REGION Network 132: FIXTURE IN UNIT 02 STATION 0 ANY CALIBRATION MISSING
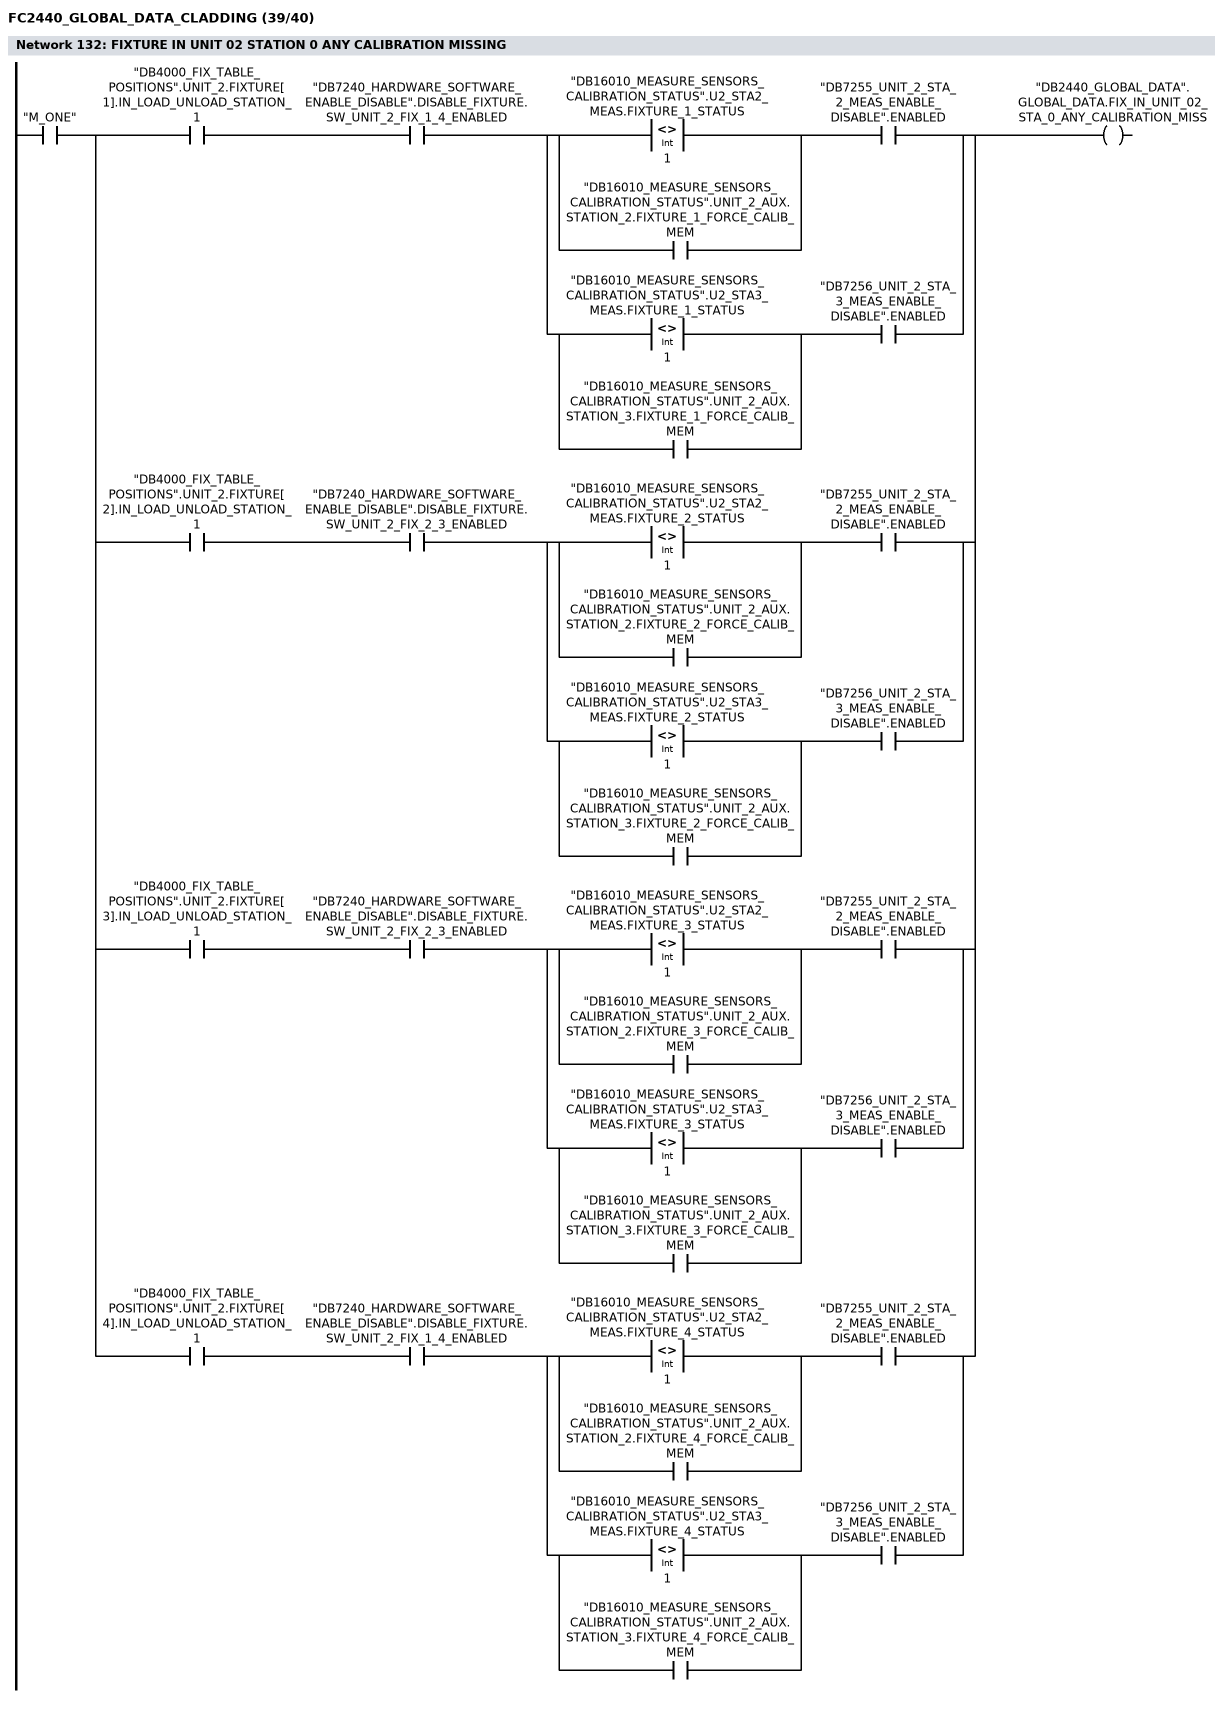
   RUNG wire#powerrail
      Contact( "M_ONE" )
      wire#w1
      Contact( "DB4000_FIX_TABLE_POSITIONS".UNIT_2.FIXTURE[1].IN_LOAD_UNLOAD_STATION_1 )
      Contact( "DB7240_HARDWARE_SOFTWARE_ENABLE_DISABLE".DISABLE_FIXTURE.SW_UNIT_2_FIX_1_4_ENABLED )
      wire#w2
      { S7_Templates := "SrcType := Int" } NE_Contact(in1 := "DB16010_MEASURE_SENSORS_CALIBRATION_STATUS".U2_STA2_MEAS.FIXTURE_1_STATUS, in2 := 1)
      wire#w3
      Contact( "DB7255_UNIT_2_STA_2_MEAS_ENABLE_DISABLE".ENABLED )
      wire#w4
      Coil( "DB2440_GLOBAL_DATA".GLOBAL_DATA.FIX_IN_UNIT_02_STA_0_ANY_CALIBRATION_MISS )
   END_RUNG
   RUNG wire#w2
      Contact( "DB16010_MEASURE_SENSORS_CALIBRATION_STATUS".UNIT_2_AUX.STATION_2.FIXTURE_1_FORCE_CALIB_MEM )
   END_RUNG wire#w3
   RUNG wire#w2
      { S7_Templates := "SrcType := Int" } NE_Contact(in1 := "DB16010_MEASURE_SENSORS_CALIBRATION_STATUS".U2_STA3_MEAS.FIXTURE_1_STATUS, in2 := 1)
      wire#w5
      Contact( "DB7256_UNIT_2_STA_3_MEAS_ENABLE_DISABLE".ENABLED )
   END_RUNG wire#w4
   RUNG wire#w2
      Contact( "DB16010_MEASURE_SENSORS_CALIBRATION_STATUS".UNIT_2_AUX.STATION_3.FIXTURE_1_FORCE_CALIB_MEM )
   END_RUNG wire#w5
   RUNG wire#w1
      Contact( "DB4000_FIX_TABLE_POSITIONS".UNIT_2.FIXTURE[2].IN_LOAD_UNLOAD_STATION_1 )
      Contact( "DB7240_HARDWARE_SOFTWARE_ENABLE_DISABLE".DISABLE_FIXTURE.SW_UNIT_2_FIX_2_3_ENABLED )
      wire#w6
      { S7_Templates := "SrcType := Int" } NE_Contact(in1 := "DB16010_MEASURE_SENSORS_CALIBRATION_STATUS".U2_STA2_MEAS.FIXTURE_2_STATUS, in2 := 1)
      wire#w7
      Contact( "DB7255_UNIT_2_STA_2_MEAS_ENABLE_DISABLE".ENABLED )
   END_RUNG wire#w4
   RUNG wire#w6
      Contact( "DB16010_MEASURE_SENSORS_CALIBRATION_STATUS".UNIT_2_AUX.STATION_2.FIXTURE_2_FORCE_CALIB_MEM )
   END_RUNG wire#w7
   RUNG wire#w6
      { S7_Templates := "SrcType := Int" } NE_Contact(in1 := "DB16010_MEASURE_SENSORS_CALIBRATION_STATUS".U2_STA3_MEAS.FIXTURE_2_STATUS, in2 := 1)
      wire#w8
      Contact( "DB7256_UNIT_2_STA_3_MEAS_ENABLE_DISABLE".ENABLED )
   END_RUNG wire#w4
   RUNG wire#w6
      Contact( "DB16010_MEASURE_SENSORS_CALIBRATION_STATUS".UNIT_2_AUX.STATION_3.FIXTURE_2_FORCE_CALIB_MEM )
   END_RUNG wire#w8
   RUNG wire#w1
      Contact( "DB4000_FIX_TABLE_POSITIONS".UNIT_2.FIXTURE[3].IN_LOAD_UNLOAD_STATION_1 )
      Contact( "DB7240_HARDWARE_SOFTWARE_ENABLE_DISABLE".DISABLE_FIXTURE.SW_UNIT_2_FIX_2_3_ENABLED )
      wire#w9
      { S7_Templates := "SrcType := Int" } NE_Contact(in1 := "DB16010_MEASURE_SENSORS_CALIBRATION_STATUS".U2_STA2_MEAS.FIXTURE_3_STATUS, in2 := 1)
      wire#w10
      Contact( "DB7255_UNIT_2_STA_2_MEAS_ENABLE_DISABLE".ENABLED )
   END_RUNG wire#w4
   RUNG wire#w9
      Contact( "DB16010_MEASURE_SENSORS_CALIBRATION_STATUS".UNIT_2_AUX.STATION_2.FIXTURE_3_FORCE_CALIB_MEM )
   END_RUNG wire#w10
   RUNG wire#w9
      { S7_Templates := "SrcType := Int" } NE_Contact(in1 := "DB16010_MEASURE_SENSORS_CALIBRATION_STATUS".U2_STA3_MEAS.FIXTURE_3_STATUS, in2 := 1)
      wire#w11
      Contact( "DB7256_UNIT_2_STA_3_MEAS_ENABLE_DISABLE".ENABLED )
   END_RUNG wire#w4
   RUNG wire#w9
      Contact( "DB16010_MEASURE_SENSORS_CALIBRATION_STATUS".UNIT_2_AUX.STATION_3.FIXTURE_3_FORCE_CALIB_MEM )
   END_RUNG wire#w11
   RUNG wire#w1
      Contact( "DB4000_FIX_TABLE_POSITIONS".UNIT_2.FIXTURE[4].IN_LOAD_UNLOAD_STATION_1 )
      Contact( "DB7240_HARDWARE_SOFTWARE_ENABLE_DISABLE".DISABLE_FIXTURE.SW_UNIT_2_FIX_1_4_ENABLED )
      wire#w12
      { S7_Templates := "SrcType := Int" } NE_Contact(in1 := "DB16010_MEASURE_SENSORS_CALIBRATION_STATUS".U2_STA2_MEAS.FIXTURE_4_STATUS, in2 := 1)
      wire#w13
      Contact( "DB7255_UNIT_2_STA_2_MEAS_ENABLE_DISABLE".ENABLED )
   END_RUNG wire#w4
   RUNG wire#w12
      Contact( "DB16010_MEASURE_SENSORS_CALIBRATION_STATUS".UNIT_2_AUX.STATION_2.FIXTURE_4_FORCE_CALIB_MEM )
   END_RUNG wire#w13
   RUNG wire#w12
      { S7_Templates := "SrcType := Int" } NE_Contact(in1 := "DB16010_MEASURE_SENSORS_CALIBRATION_STATUS".U2_STA3_MEAS.FIXTURE_4_STATUS, in2 := 1)
      wire#w14
      Contact( "DB7256_UNIT_2_STA_3_MEAS_ENABLE_DISABLE".ENABLED )
   END_RUNG wire#w4
   RUNG wire#w12
      Contact( "DB16010_MEASURE_SENSORS_CALIBRATION_STATUS".UNIT_2_AUX.STATION_3.FIXTURE_4_FORCE_CALIB_MEM )
   END_RUNG wire#w14
   // the same network as SCL:
   "DB2440_GLOBAL_DATA".GLOBAL_DATA.FIX_IN_UNIT_02_STA_0_ANY_CALIBRATION_MISS := "M_ONE" AND (("DB4000_FIX_TABLE_POSITIONS".UNIT_2.FIXTURE[1].IN_LOAD_UNLOAD_STATION_1 AND "DB7240_HARDWARE_SOFTWARE_ENABLE_DISABLE".DISABLE_FIXTURE.SW_UNIT_2_FIX_1_4_ENABLED AND (((("DB16010_MEASURE_SENSORS_CALIBRATION_STATUS".U2_STA2_MEAS.FIXTURE_1_STATUS <> 1) OR "DB16010_MEASURE_SENSORS_CALIBRATION_STATUS".UNIT_2_AUX.STATION_2.FIXTURE_1_FORCE_CALIB_MEM) AND "DB7255_UNIT_2_STA_2_MEAS_ENABLE_DISABLE".ENABLED) OR ((("DB16010_MEASURE_SENSORS_CALIBRATION_STATUS".U2_STA3_MEAS.FIXTURE_1_STATUS <> 1) OR "DB16010_MEASURE_SENSORS_CALIBRATION_STATUS".UNIT_2_AUX.STATION_3.FIXTURE_1_FORCE_CALIB_MEM) AND "DB7256_UNIT_2_STA_3_MEAS_ENABLE_DISABLE".ENABLED))) OR ("DB4000_FIX_TABLE_POSITIONS".UNIT_2.FIXTURE[2].IN_LOAD_UNLOAD_STATION_1 AND "DB7240_HARDWARE_SOFTWARE_ENABLE_DISABLE".DISABLE_FIXTURE.SW_UNIT_2_FIX_2_3_ENABLED AND (((("DB16010_MEASURE_SENSORS_CALIBRATION_STATUS".U2_STA2_MEAS.FIXTURE_2_STATUS <> 1) OR "DB16010_MEASURE_SENSORS_CALIBRATION_STATUS".UNIT_2_AUX.STATION_2.FIXTURE_2_FORCE_CALIB_MEM) AND "DB7255_UNIT_2_STA_2_MEAS_ENABLE_DISABLE".ENABLED) OR ((("DB16010_MEASURE_SENSORS_CALIBRATION_STATUS".U2_STA3_MEAS.FIXTURE_2_STATUS <> 1) OR "DB16010_MEASURE_SENSORS_CALIBRATION_STATUS".UNIT_2_AUX.STATION_3.FIXTURE_2_FORCE_CALIB_MEM) AND "DB7256_UNIT_2_STA_3_MEAS_ENABLE_DISABLE".ENABLED))) OR ("DB4000_FIX_TABLE_POSITIONS".UNIT_2.FIXTURE[3].IN_LOAD_UNLOAD_STATION_1 AND "DB7240_HARDWARE_SOFTWARE_ENABLE_DISABLE".DISABLE_FIXTURE.SW_UNIT_2_FIX_2_3_ENABLED AND (((("DB16010_MEASURE_SENSORS_CALIBRATION_STATUS".U2_STA2_MEAS.FIXTURE_3_STATUS <> 1) OR "DB16010_MEASURE_SENSORS_CALIBRATION_STATUS".UNIT_2_AUX.STATION_2.FIXTURE_3_FORCE_CALIB_MEM) AND "DB7255_UNIT_2_STA_2_MEAS_ENABLE_DISABLE".ENABLED) OR ((("DB16010_MEASURE_SENSORS_CALIBRATION_STATUS".U2_STA3_MEAS.FIXTURE_3_STATUS <> 1) OR "DB16010_MEASURE_SENSORS_CALIBRATION_STATUS".UNIT_2_AUX.STATION_3.FIXTURE_3_FORCE_CALIB_MEM) AND "DB7256_UNIT_2_STA_3_MEAS_ENABLE_DISABLE".ENABLED))) OR ("DB4000_FIX_TABLE_POSITIONS".UNIT_2.FIXTURE[4].IN_LOAD_UNLOAD_STATION_1 AND "DB7240_HARDWARE_SOFTWARE_ENABLE_DISABLE".DISABLE_FIXTURE.SW_UNIT_2_FIX_1_4_ENABLED AND (((("DB16010_MEASURE_SENSORS_CALIBRATION_STATUS".U2_STA2_MEAS.FIXTURE_4_STATUS <> 1) OR "DB16010_MEASURE_SENSORS_CALIBRATION_STATUS".UNIT_2_AUX.STATION_2.FIXTURE_4_FORCE_CALIB_MEM) AND "DB7255_UNIT_2_STA_2_MEAS_ENABLE_DISABLE".ENABLED) OR ((("DB16010_MEASURE_SENSORS_CALIBRATION_STATUS".U2_STA3_MEAS.FIXTURE_4_STATUS <> 1) OR "DB16010_MEASURE_SENSORS_CALIBRATION_STATUS".UNIT_2_AUX.STATION_3.FIXTURE_4_FORCE_CALIB_MEM) AND "DB7256_UNIT_2_STA_3_MEAS_ENABLE_DISABLE".ENABLED))));
END_REGION

REGION Network 133: UNIT 01 ANY FIXTURE CALIBRATION MISSING
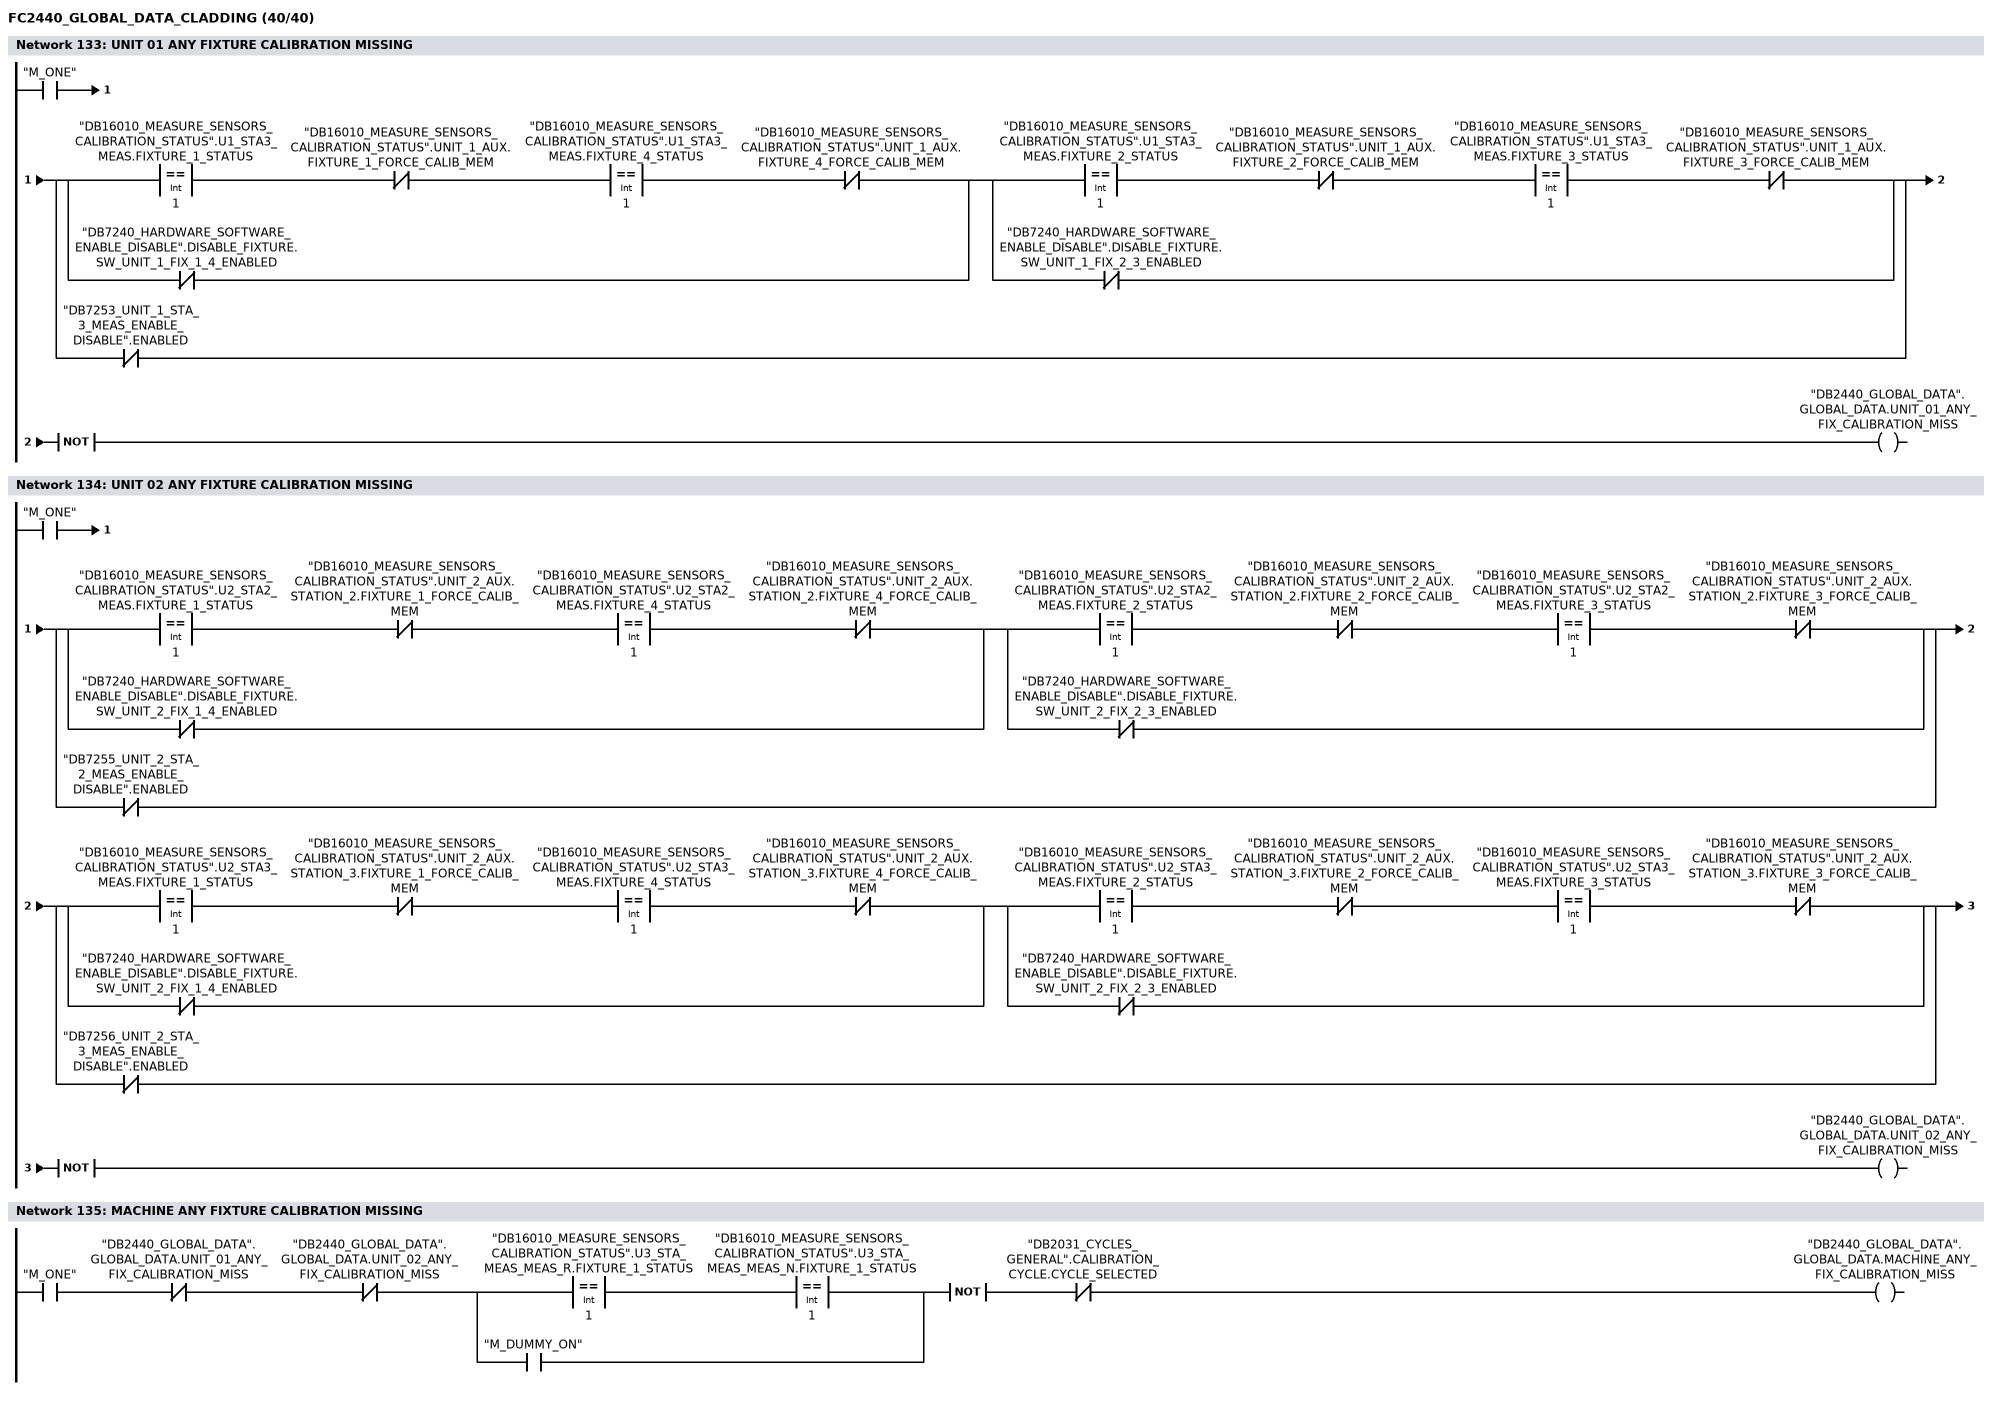
   RUNG wire#powerrail
      Contact( "M_ONE" )
      wire#w1
      { S7_Templates := "SrcType := Int" } EQ_Contact(in1 := "DB16010_MEASURE_SENSORS_CALIBRATION_STATUS".U1_STA3_MEAS.FIXTURE_1_STATUS, in2 := 1)
      I_Contact( "DB16010_MEASURE_SENSORS_CALIBRATION_STATUS".UNIT_1_AUX.FIXTURE_1_FORCE_CALIB_MEM )
      { S7_Templates := "SrcType := Int" } EQ_Contact(in1 := "DB16010_MEASURE_SENSORS_CALIBRATION_STATUS".U1_STA3_MEAS.FIXTURE_4_STATUS, in2 := 1)
      I_Contact( "DB16010_MEASURE_SENSORS_CALIBRATION_STATUS".UNIT_1_AUX.FIXTURE_4_FORCE_CALIB_MEM )
      wire#w2
      { S7_Templates := "SrcType := Int" } EQ_Contact(in1 := "DB16010_MEASURE_SENSORS_CALIBRATION_STATUS".U1_STA3_MEAS.FIXTURE_2_STATUS, in2 := 1)
      I_Contact( "DB16010_MEASURE_SENSORS_CALIBRATION_STATUS".UNIT_1_AUX.FIXTURE_2_FORCE_CALIB_MEM )
      { S7_Templates := "SrcType := Int" } EQ_Contact(in1 := "DB16010_MEASURE_SENSORS_CALIBRATION_STATUS".U1_STA3_MEAS.FIXTURE_3_STATUS, in2 := 1)
      I_Contact( "DB16010_MEASURE_SENSORS_CALIBRATION_STATUS".UNIT_1_AUX.FIXTURE_3_FORCE_CALIB_MEM )
      wire#w3
      Not()
      Coil( "DB2440_GLOBAL_DATA".GLOBAL_DATA.UNIT_01_ANY_FIX_CALIBRATION_MISS )
   END_RUNG
   RUNG wire#w1
      I_Contact( "DB7240_HARDWARE_SOFTWARE_ENABLE_DISABLE".DISABLE_FIXTURE.SW_UNIT_1_FIX_1_4_ENABLED )
   END_RUNG wire#w2
   RUNG wire#w2
      I_Contact( "DB7240_HARDWARE_SOFTWARE_ENABLE_DISABLE".DISABLE_FIXTURE.SW_UNIT_1_FIX_2_3_ENABLED )
   END_RUNG wire#w3
   RUNG wire#w1
      I_Contact( "DB7253_UNIT_1_STA_3_MEAS_ENABLE_DISABLE".ENABLED )
   END_RUNG wire#w3
   // the same network as SCL:
   "DB2440_GLOBAL_DATA".GLOBAL_DATA.UNIT_01_ANY_FIX_CALIBRATION_MISS := NOT ("M_ONE" AND ((((("DB16010_MEASURE_SENSORS_CALIBRATION_STATUS".U1_STA3_MEAS.FIXTURE_1_STATUS = 1) AND NOT "DB16010_MEASURE_SENSORS_CALIBRATION_STATUS".UNIT_1_AUX.FIXTURE_1_FORCE_CALIB_MEM AND ("DB16010_MEASURE_SENSORS_CALIBRATION_STATUS".U1_STA3_MEAS.FIXTURE_4_STATUS = 1) AND NOT "DB16010_MEASURE_SENSORS_CALIBRATION_STATUS".UNIT_1_AUX.FIXTURE_4_FORCE_CALIB_MEM) OR NOT "DB7240_HARDWARE_SOFTWARE_ENABLE_DISABLE".DISABLE_FIXTURE.SW_UNIT_1_FIX_1_4_ENABLED) AND ((("DB16010_MEASURE_SENSORS_CALIBRATION_STATUS".U1_STA3_MEAS.FIXTURE_2_STATUS = 1) AND NOT "DB16010_MEASURE_SENSORS_CALIBRATION_STATUS".UNIT_1_AUX.FIXTURE_2_FORCE_CALIB_MEM AND ("DB16010_MEASURE_SENSORS_CALIBRATION_STATUS".U1_STA3_MEAS.FIXTURE_3_STATUS = 1) AND NOT "DB16010_MEASURE_SENSORS_CALIBRATION_STATUS".UNIT_1_AUX.FIXTURE_3_FORCE_CALIB_MEM) OR NOT "DB7240_HARDWARE_SOFTWARE_ENABLE_DISABLE".DISABLE_FIXTURE.SW_UNIT_1_FIX_2_3_ENABLED)) OR NOT "DB7253_UNIT_1_STA_3_MEAS_ENABLE_DISABLE".ENABLED));
END_REGION

REGION Network 134: UNIT 02 ANY FIXTURE CALIBRATION MISSING
   RUNG wire#powerrail
      Contact( "M_ONE" )
      wire#w1
      { S7_Templates := "SrcType := Int" } EQ_Contact(in1 := "DB16010_MEASURE_SENSORS_CALIBRATION_STATUS".U2_STA2_MEAS.FIXTURE_1_STATUS, in2 := 1)
      I_Contact( "DB16010_MEASURE_SENSORS_CALIBRATION_STATUS".UNIT_2_AUX.STATION_2.FIXTURE_1_FORCE_CALIB_MEM )
      { S7_Templates := "SrcType := Int" } EQ_Contact(in1 := "DB16010_MEASURE_SENSORS_CALIBRATION_STATUS".U2_STA2_MEAS.FIXTURE_4_STATUS, in2 := 1)
      I_Contact( "DB16010_MEASURE_SENSORS_CALIBRATION_STATUS".UNIT_2_AUX.STATION_2.FIXTURE_4_FORCE_CALIB_MEM )
      wire#w2
      { S7_Templates := "SrcType := Int" } EQ_Contact(in1 := "DB16010_MEASURE_SENSORS_CALIBRATION_STATUS".U2_STA2_MEAS.FIXTURE_2_STATUS, in2 := 1)
      I_Contact( "DB16010_MEASURE_SENSORS_CALIBRATION_STATUS".UNIT_2_AUX.STATION_2.FIXTURE_2_FORCE_CALIB_MEM )
      { S7_Templates := "SrcType := Int" } EQ_Contact(in1 := "DB16010_MEASURE_SENSORS_CALIBRATION_STATUS".U2_STA2_MEAS.FIXTURE_3_STATUS, in2 := 1)
      I_Contact( "DB16010_MEASURE_SENSORS_CALIBRATION_STATUS".UNIT_2_AUX.STATION_2.FIXTURE_3_FORCE_CALIB_MEM )
      wire#w3
      { S7_Templates := "SrcType := Int" } EQ_Contact(in1 := "DB16010_MEASURE_SENSORS_CALIBRATION_STATUS".U2_STA3_MEAS.FIXTURE_1_STATUS, in2 := 1)
      I_Contact( "DB16010_MEASURE_SENSORS_CALIBRATION_STATUS".UNIT_2_AUX.STATION_3.FIXTURE_1_FORCE_CALIB_MEM )
      { S7_Templates := "SrcType := Int" } EQ_Contact(in1 := "DB16010_MEASURE_SENSORS_CALIBRATION_STATUS".U2_STA3_MEAS.FIXTURE_4_STATUS, in2 := 1)
      I_Contact( "DB16010_MEASURE_SENSORS_CALIBRATION_STATUS".UNIT_2_AUX.STATION_3.FIXTURE_4_FORCE_CALIB_MEM )
      wire#w4
      { S7_Templates := "SrcType := Int" } EQ_Contact(in1 := "DB16010_MEASURE_SENSORS_CALIBRATION_STATUS".U2_STA3_MEAS.FIXTURE_2_STATUS, in2 := 1)
      I_Contact( "DB16010_MEASURE_SENSORS_CALIBRATION_STATUS".UNIT_2_AUX.STATION_3.FIXTURE_2_FORCE_CALIB_MEM )
      { S7_Templates := "SrcType := Int" } EQ_Contact(in1 := "DB16010_MEASURE_SENSORS_CALIBRATION_STATUS".U2_STA3_MEAS.FIXTURE_3_STATUS, in2 := 1)
      I_Contact( "DB16010_MEASURE_SENSORS_CALIBRATION_STATUS".UNIT_2_AUX.STATION_3.FIXTURE_3_FORCE_CALIB_MEM )
      wire#w5
      Not()
      Coil( "DB2440_GLOBAL_DATA".GLOBAL_DATA.UNIT_02_ANY_FIX_CALIBRATION_MISS )
   END_RUNG
   RUNG wire#w1
      I_Contact( "DB7240_HARDWARE_SOFTWARE_ENABLE_DISABLE".DISABLE_FIXTURE.SW_UNIT_2_FIX_1_4_ENABLED )
   END_RUNG wire#w2
   RUNG wire#w2
      I_Contact( "DB7240_HARDWARE_SOFTWARE_ENABLE_DISABLE".DISABLE_FIXTURE.SW_UNIT_2_FIX_2_3_ENABLED )
   END_RUNG wire#w3
   RUNG wire#w1
      I_Contact( "DB7255_UNIT_2_STA_2_MEAS_ENABLE_DISABLE".ENABLED )
   END_RUNG wire#w3
   RUNG wire#w3
      I_Contact( "DB7240_HARDWARE_SOFTWARE_ENABLE_DISABLE".DISABLE_FIXTURE.SW_UNIT_2_FIX_1_4_ENABLED )
   END_RUNG wire#w4
   RUNG wire#w4
      I_Contact( "DB7240_HARDWARE_SOFTWARE_ENABLE_DISABLE".DISABLE_FIXTURE.SW_UNIT_2_FIX_2_3_ENABLED )
   END_RUNG wire#w5
   RUNG wire#w3
      I_Contact( "DB7256_UNIT_2_STA_3_MEAS_ENABLE_DISABLE".ENABLED )
   END_RUNG wire#w5
   // the same network as SCL:
   "DB2440_GLOBAL_DATA".GLOBAL_DATA.UNIT_02_ANY_FIX_CALIBRATION_MISS := NOT ("M_ONE" AND ((((("DB16010_MEASURE_SENSORS_CALIBRATION_STATUS".U2_STA2_MEAS.FIXTURE_1_STATUS = 1) AND NOT "DB16010_MEASURE_SENSORS_CALIBRATION_STATUS".UNIT_2_AUX.STATION_2.FIXTURE_1_FORCE_CALIB_MEM AND ("DB16010_MEASURE_SENSORS_CALIBRATION_STATUS".U2_STA2_MEAS.FIXTURE_4_STATUS = 1) AND NOT "DB16010_MEASURE_SENSORS_CALIBRATION_STATUS".UNIT_2_AUX.STATION_2.FIXTURE_4_FORCE_CALIB_MEM) OR NOT "DB7240_HARDWARE_SOFTWARE_ENABLE_DISABLE".DISABLE_FIXTURE.SW_UNIT_2_FIX_1_4_ENABLED) AND ((("DB16010_MEASURE_SENSORS_CALIBRATION_STATUS".U2_STA2_MEAS.FIXTURE_2_STATUS = 1) AND NOT "DB16010_MEASURE_SENSORS_CALIBRATION_STATUS".UNIT_2_AUX.STATION_2.FIXTURE_2_FORCE_CALIB_MEM AND ("DB16010_MEASURE_SENSORS_CALIBRATION_STATUS".U2_STA2_MEAS.FIXTURE_3_STATUS = 1) AND NOT "DB16010_MEASURE_SENSORS_CALIBRATION_STATUS".UNIT_2_AUX.STATION_2.FIXTURE_3_FORCE_CALIB_MEM) OR NOT "DB7240_HARDWARE_SOFTWARE_ENABLE_DISABLE".DISABLE_FIXTURE.SW_UNIT_2_FIX_2_3_ENABLED)) OR NOT "DB7255_UNIT_2_STA_2_MEAS_ENABLE_DISABLE".ENABLED) AND ((((("DB16010_MEASURE_SENSORS_CALIBRATION_STATUS".U2_STA3_MEAS.FIXTURE_1_STATUS = 1) AND NOT "DB16010_MEASURE_SENSORS_CALIBRATION_STATUS".UNIT_2_AUX.STATION_3.FIXTURE_1_FORCE_CALIB_MEM AND ("DB16010_MEASURE_SENSORS_CALIBRATION_STATUS".U2_STA3_MEAS.FIXTURE_4_STATUS = 1) AND NOT "DB16010_MEASURE_SENSORS_CALIBRATION_STATUS".UNIT_2_AUX.STATION_3.FIXTURE_4_FORCE_CALIB_MEM) OR NOT "DB7240_HARDWARE_SOFTWARE_ENABLE_DISABLE".DISABLE_FIXTURE.SW_UNIT_2_FIX_1_4_ENABLED) AND ((("DB16010_MEASURE_SENSORS_CALIBRATION_STATUS".U2_STA3_MEAS.FIXTURE_2_STATUS = 1) AND NOT "DB16010_MEASURE_SENSORS_CALIBRATION_STATUS".UNIT_2_AUX.STATION_3.FIXTURE_2_FORCE_CALIB_MEM AND ("DB16010_MEASURE_SENSORS_CALIBRATION_STATUS".U2_STA3_MEAS.FIXTURE_3_STATUS = 1) AND NOT "DB16010_MEASURE_SENSORS_CALIBRATION_STATUS".UNIT_2_AUX.STATION_3.FIXTURE_3_FORCE_CALIB_MEM) OR NOT "DB7240_HARDWARE_SOFTWARE_ENABLE_DISABLE".DISABLE_FIXTURE.SW_UNIT_2_FIX_2_3_ENABLED)) OR NOT "DB7256_UNIT_2_STA_3_MEAS_ENABLE_DISABLE".ENABLED));
END_REGION

REGION Network 135: MACHINE ANY FIXTURE CALIBRATION MISSING
   RUNG wire#powerrail
      Contact( "M_ONE" )
      I_Contact( "DB2440_GLOBAL_DATA".GLOBAL_DATA.UNIT_01_ANY_FIX_CALIBRATION_MISS )
      I_Contact( "DB2440_GLOBAL_DATA".GLOBAL_DATA.UNIT_02_ANY_FIX_CALIBRATION_MISS )
      wire#w1
      { S7_Templates := "SrcType := Int" } EQ_Contact(in1 := "DB16010_MEASURE_SENSORS_CALIBRATION_STATUS".U3_STA_MEAS_MEAS_R.FIXTURE_1_STATUS, in2 := 1)
      { S7_Templates := "SrcType := Int" } EQ_Contact(in1 := "DB16010_MEASURE_SENSORS_CALIBRATION_STATUS".U3_STA_MEAS_MEAS_N.FIXTURE_1_STATUS, in2 := 1)
      wire#w2
      Not()
      I_Contact( "DB2031_CYCLES_GENERAL".CALIBRATION_CYCLE.CYCLE_SELECTED )
      Coil( "DB2440_GLOBAL_DATA".GLOBAL_DATA.MACHINE_ANY_FIX_CALIBRATION_MISS )
   END_RUNG
   RUNG wire#w1
      Contact( "M_DUMMY_ON" )
   END_RUNG wire#w2
   // the same network as SCL:
   "DB2440_GLOBAL_DATA".GLOBAL_DATA.MACHINE_ANY_FIX_CALIBRATION_MISS := NOT ("M_ONE" AND NOT "DB2440_GLOBAL_DATA".GLOBAL_DATA.UNIT_01_ANY_FIX_CALIBRATION_MISS AND NOT "DB2440_GLOBAL_DATA".GLOBAL_DATA.UNIT_02_ANY_FIX_CALIBRATION_MISS AND ((("DB16010_MEASURE_SENSORS_CALIBRATION_STATUS".U3_STA_MEAS_MEAS_R.FIXTURE_1_STATUS = 1) AND ("DB16010_MEASURE_SENSORS_CALIBRATION_STATUS".U3_STA_MEAS_MEAS_N.FIXTURE_1_STATUS = 1)) OR "M_DUMMY_ON")) AND NOT "DB2031_CYCLES_GENERAL".CALIBRATION_CYCLE.CYCLE_SELECTED;
END_REGION
END_FUNCTION
